// SIMATIC STEP 7 (V5.x) project RLI-p1
// CPU: CPU 412-1
// CPU: CPU 412-1
// station: Matériel
// station: Maitre
// station: P_ADR_BUS
// station: P_ADR_BUS
// station: Matériel
// station: Esclave
// program: Programme S7(1)
// program: Programme S7(1)

DATA_BLOCK DB 10
VERSION : 0.1
  STRUCT
   DB_VAR : INT  := 1;	//Variable temporaire de réservation
   var2 : INT  := 2;
   Var3 : INT  := 3;
   var4 : INT  := 4;
   VAR5 : INT  := 5;
   Var6 : INT  := 6;
  END_STRUCT ;	
BEGIN
   DB_VAR := 1;
   var2 := 2;
   Var3 := 3;
   var4 := 4;
   VAR5 := 5;
   Var6 := 6;
END_DATA_BLOCK

ORGANIZATION_BLOCK OB 1
TITLE = "Main Program Sweep (Cycle)"
VERSION : 0.1
VAR_TEMP
  OB1_EV_CLASS : BYTE ;	//Bits 0-3 = 1 (Coming event), Bits 4-7 = 1 (Event class 1)
  OB1_SCAN_1 : BYTE ;	//1 (Cold restart scan 1 of OB 1), 3 (Scan 2-n of OB 1)
  OB1_PRIORITY : BYTE ;	//Priority of OB Execution
  OB1_OB_NUMBR : BYTE ;	//1 (Organization block 1, OB1)
  OB1_RESERVED_1 : BYTE ;	//Reserved for system
  OB1_RESERVED_2 : BYTE ;	//Reserved for system
  OB1_PREV_CYCLE : INT ;	//Cycle time of previous OB1 scan (milliseconds)
  OB1_MIN_CYCLE : INT ;	//Minimum cycle time of OB1 (milliseconds)
  OB1_MAX_CYCLE : INT ;	//Maximum cycle time of OB1 (milliseconds)
  OB1_DATE_TIME : DATE_AND_TIME ;	//Date and time OB1 started
END_VAR
BEGIN
// (block stored without names or comments; labels and parameter names are numbered)
END_ORGANIZATION_BLOCK

DATA_BLOCK DB 15
VERSION : 0.1
  STRUCT
   DB_VAR : INT ;	//Variable temporaire de réservation
   VAr1 : INT ;
   VAR2 : INT ;
   var3 : INT ;
   VAr4 : INT ;
   VAr5 : INT ;
   VAr56 : INT ;
   VAr7 : INT ;
  END_STRUCT ;	
BEGIN
   var3 := 4;
END_DATA_BLOCK

ORGANIZATION_BLOCK OB 1
TITLE = "Main Program Sweep (Cycle)"
VERSION : 0.1
VAR_TEMP
  OB1_EV_CLASS : BYTE ;	//Bits 0-3 = 1 (Coming event), Bits 4-7 = 1 (Event class 1)
  OB1_SCAN_1 : BYTE ;	//1 (Cold restart scan 1 of OB 1), 3 (Scan 2-n of OB 1)
  OB1_PRIORITY : BYTE ;	//Priority of OB Execution
  OB1_OB_NUMBR : BYTE ;	//1 (Organization block 1, OB1)
  OB1_RESERVED_1 : BYTE ;	//Reserved for system
  OB1_RESERVED_2 : BYTE ;	//Reserved for system
  OB1_PREV_CYCLE : INT ;	//Cycle time of previous OB1 scan (milliseconds)
  OB1_MIN_CYCLE : INT ;	//Minimum cycle time of OB1 (milliseconds)
  OB1_MAX_CYCLE : INT ;	//Maximum cycle time of OB1 (milliseconds)
  OB1_DATE_TIME : DATE_AND_TIME ;	//Date and time OB1 started
END_VAR
BEGIN
// (block stored without names or comments; labels and parameter names are numbered)
END_ORGANIZATION_BLOCK
